// TIA Portal project "ControlPID_FactoryIO" (V16)

(* hardware
DEVICE "S7-1200 station_1"  S7-1200 Station
   slot 0: "Rack_0"  S7-1200 Rack  Rack  V1.0
   slot 1: "PLC_1"  CPU 1214C AC/DC/Rly  6ES7 214-1BG40-0XB0  V4.4
DEVICE "HMI_1"  TP1200 Comfort
   slot 0: "HMI_1"  TP1200 Comfort  6AV2 124-0MC01-0AX0  16.0.0.0
   slot 1: "HMI_RT_1"  TP1200 Comfort  6AV2 124-0MC01-0AX0  16.0.0.0
   slot 5: "HMI_1.IE_CP_1"  PROFINET Interface  16.0.0.0
      slot 1: "PROFINET Interface_1"  PROFINET Interface
         slot 1: "Port_1"  Port
         slot 2: "Port_2"  Port
   slot 7: "HMI_1.MPI/DP_CP_1"  MPI/DP Interface  16.0.0.0
*)

// ===== PLC "PLC_1"  CPU 1214C AC/DC/Rly =====

VAR_GLOBAL   // PLC tag table "Default tag table"
   "Start" AT %I20.0 : Bool;
   "Stop" AT %I20.1 : Bool;
   "Led" AT %Q0.0 : Bool;
   "SP" AT %IW100 : Int;
   "Level Sensor" AT %IW102 : Int;
   "Fill Valve" AT %QW100 : Int;
   "Discharge Valve" AT %QW102 : Int;
   "Display SP" AT %QW104 : Int;
   "Display PV" AT %QW106 : Int;
   "SP(mm)" AT %MD10 : Real;
   "SP(%)" AT %MD14 : Real;
   "PV(mm)" AT %MD18 : Real;
   "PV(%)" AT %MD22 : Real;
   "CV(%)" AT %MD26 : Real;
END_VAR

DATA_BLOCK "Set Point_DB"   // DB1
{ S7_Optimized_Access := 'TRUE' }
VERSION : 0.1
// stored: InstanceOfName Set Point
"Set Point"
BEGIN
END_DATA_BLOCK

DATA_BLOCK "Sensor_DB"   // DB2
{ S7_Optimized_Access := 'TRUE' }
VERSION : 0.1
// stored: InstanceOfName Sensor
"Sensor"
BEGIN
END_DATA_BLOCK

DATA_BLOCK "Output PID_DB"   // DB3
{ S7_Optimized_Access := 'TRUE' }
VERSION : 0.1
// stored: InstanceOfName Output PID
"Output PID"
BEGIN
END_DATA_BLOCK

FUNCTION_BLOCK "Set Point"   // FB1, LAD
{ S7_Optimized_Access := 'TRUE' }
VERSION : 0.1
   VAR_INPUT
      InAnalog : Int;
      LevelMax : Real;
   END_VAR
   VAR_OUTPUT
      "Level(mm)" : Real;
      "Level(%)" : Real;
   END_VAR
   VAR
      Cal : Real;
   END_VAR
BEGIN

REGION Network 1
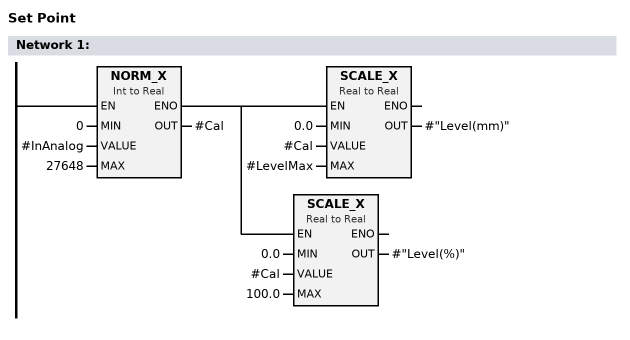
   RUNG wire#powerrail
      { S7_Templates := "[SrcType := Int, DestType := Real]" } Normalize(min := 0, value := #InAnalog, max := 27648, out => #Cal)
      wire#w1
      { S7_Templates := "[SrcType := Real, DestType := Real]" } Scale(min := 0.0, value := #Cal, max := #LevelMax, out => #"Level(mm)")
   END_RUNG
   RUNG wire#w1
      { S7_Templates := "[SrcType := Real, DestType := Real]" } Scale(min := 0.0, value := #Cal, max := 100.0, out => #"Level(%)")
   END_RUNG
   // the same network as SCL:
   #Cal := NORM_X(MIN := 0, VALUE := #InAnalog, MAX := 27648);
   #"Level(mm)" := SCALE_X(MIN := 0.0, VALUE := #Cal, MAX := #LevelMax);
   #"Level(%)" := SCALE_X(MIN := 0.0, VALUE := #Cal, MAX := 100.0);
END_REGION
END_FUNCTION_BLOCK

FUNCTION_BLOCK "Sensor"   // FB2, LAD
{ S7_Optimized_Access := 'TRUE' }
VERSION : 0.1
   VAR_INPUT
      InAnalog : Int;
      LevelMax : Real;
   END_VAR
   VAR_OUTPUT
      "Level(mm)" : Real;
      "Level(%)" : Real;
   END_VAR
   VAR
      Cal : Real;
   END_VAR
BEGIN

REGION Network 1
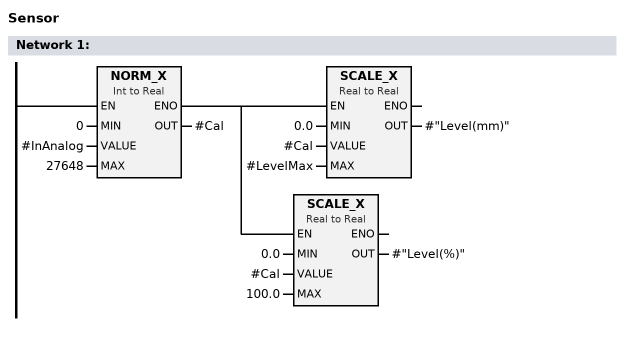
   RUNG wire#powerrail
      { S7_Templates := "[SrcType := Int, DestType := Real]" } Normalize(min := 0, value := #InAnalog, max := 27648, out => #Cal)
      wire#w1
      { S7_Templates := "[SrcType := Real, DestType := Real]" } Scale(min := 0.0, value := #Cal, max := #LevelMax, out => #"Level(mm)")
   END_RUNG
   RUNG wire#w1
      { S7_Templates := "[SrcType := Real, DestType := Real]" } Scale(min := 0.0, value := #Cal, max := 100.0, out => #"Level(%)")
   END_RUNG
   // the same network as SCL:
   #Cal := NORM_X(MIN := 0, VALUE := #InAnalog, MAX := 27648);
   #"Level(mm)" := SCALE_X(MIN := 0.0, VALUE := #Cal, MAX := #LevelMax);
   #"Level(%)" := SCALE_X(MIN := 0.0, VALUE := #Cal, MAX := 100.0);
END_REGION
END_FUNCTION_BLOCK

FUNCTION_BLOCK "Output PID"   // FB3, LAD
{ S7_Optimized_Access := 'TRUE' }
VERSION : 0.1
   VAR_INPUT
      OutputPID : Real;
   END_VAR
   VAR_OUTPUT
      V_Full : Int;
      V_Emty : Int;
   END_VAR
   VAR
      OutputPID_Cal : Real;
      Cal : Real;
      Out_Value : Int;
   END_VAR
BEGIN

REGION Network 1
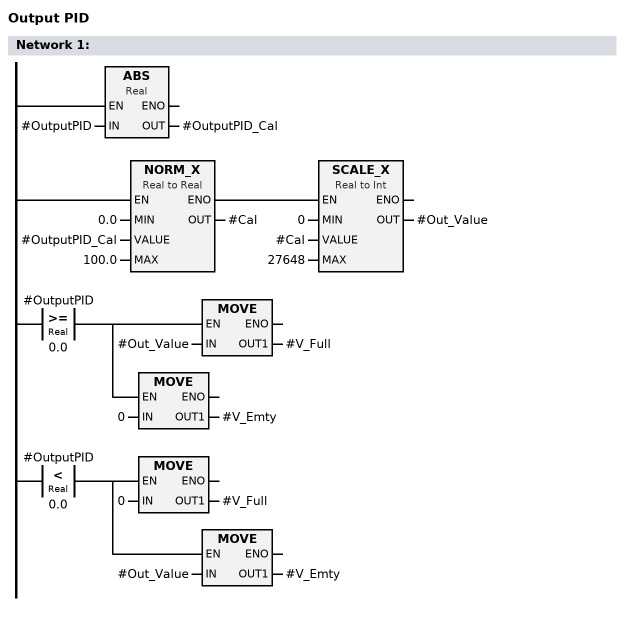
   RUNG wire#powerrail
      { S7_Templates := "SrcType := Real" } Abs(in := #OutputPID, out => #OutputPID_Cal)
   END_RUNG
   RUNG wire#powerrail
      { S7_Templates := "[SrcType := Real, DestType := Real]" } Normalize(min := 0.0, value := #OutputPID_Cal, max := 100.0, out => #Cal)
      { S7_Templates := "[SrcType := Real, DestType := Int]" } Scale(min := 0, value := #Cal, max := 27648, out => #Out_Value)
   END_RUNG
   RUNG wire#powerrail
      { S7_Templates := "SrcType := Real" } GE_Contact(in1 := #OutputPID, in2 := 0.0)
      wire#w1
      Move(in := #Out_Value, out1 => #V_Full)
   END_RUNG
   RUNG wire#w1
      Move(in := 0, out1 => #V_Emty)
   END_RUNG
   RUNG wire#powerrail
      { S7_Templates := "SrcType := Real" } LT_Contact(in1 := #OutputPID, in2 := 0.0)
      wire#w2
      Move(in := 0, out1 => #V_Full)
   END_RUNG
   RUNG wire#w2
      Move(in := #Out_Value, out1 => #V_Emty)
   END_RUNG
   // the same network as SCL:
   #OutputPID_Cal := ABS(#OutputPID);
   #Cal := NORM_X(MIN := 0.0, VALUE := #OutputPID_Cal, MAX := 100.0);
   #Out_Value := SCALE_X(MIN := 0, VALUE := #Cal, MAX := 27648);
   IF #OutputPID >= 0.0 THEN
       #V_Full := #Out_Value;
       #V_Emty := 0;
   END_IF;
   IF #OutputPID < 0.0 THEN
       #V_Full := 0;
       #V_Emty := #Out_Value;
   END_IF;
END_REGION
END_FUNCTION_BLOCK

ORGANIZATION_BLOCK "Main"   // OB1, LAD, ProgramCycle
TITLE = "Main Program Sweep (Cycle)"
{ S7_Optimized_Access := 'TRUE' }
VERSION : 0.1
   VAR_INPUT
      Initial_Call : Bool;   // Initial call of this OB
      Remanence : Bool;   // =True, if remanent data are available
   END_VAR
   VAR_TEMP   // added for the SCL form of the ladder/FBD networks
      _w1 : Bool;
      _w2 : Bool;
   END_VAR
BEGIN

REGION Network 1
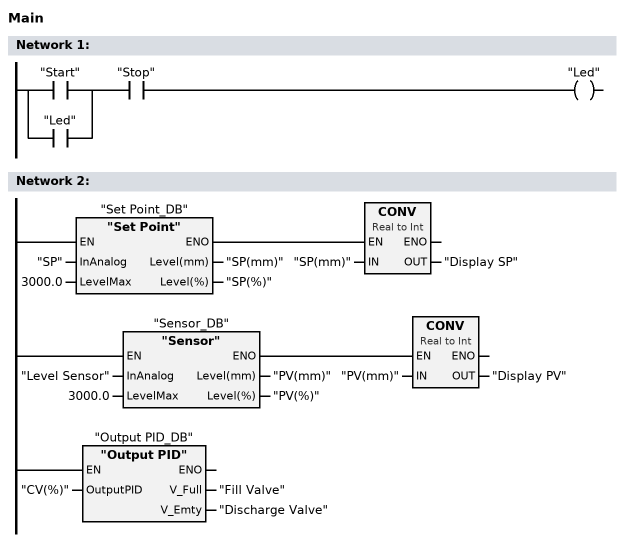
   RUNG wire#powerrail
      Contact( "Start" )
      wire#w1
      Contact( "Stop" )
      Coil( "Led" )
   END_RUNG
   RUNG wire#powerrail
      Contact( "Led" )
   END_RUNG wire#w1
   // the same network as SCL:
   "Led" := ("Start" OR "Led") AND "Stop";
END_REGION

REGION Network 2
   RUNG wire#powerrail
      "Set Point_DB"(InAnalog := "SP", LevelMax := 3000.0, "Level(mm)" => "SP(mm)", "Level(%)" => "SP(%)")
      { S7_Templates := "[SrcType := Real, DestType := Int]" } Convert(in := "SP(mm)", out => "Display SP")
   END_RUNG
   RUNG wire#powerrail
      "Sensor_DB"(InAnalog := "Level Sensor", LevelMax := 3000.0, "Level(mm)" => "PV(mm)", "Level(%)" => "PV(%)")
      { S7_Templates := "[SrcType := Real, DestType := Int]" } Convert(in := "PV(mm)", out => "Display PV")
   END_RUNG
   RUNG wire#powerrail
      "Output PID_DB"(OutputPID := "CV(%)", V_Full => "Fill Valve", V_Emty => "Discharge Valve")
   END_RUNG
   // the same network as SCL:
   "Set Point_DB"(InAnalog := "SP",   // "Set Point"
                  LevelMax := 3000.0,
                  "Level(mm)" => "SP(mm)",
                  "Level(%)" => "SP(%)",
                  ENO => #_w1);
   IF #_w1 THEN "Display SP" := REAL_TO_INT("SP(mm)"); END_IF;
   "Sensor_DB"(InAnalog := "Level Sensor",   // "Sensor"
               LevelMax := 3000.0,
               "Level(mm)" => "PV(mm)",
               "Level(%)" => "PV(%)",
               ENO => #_w2);
   IF #_w2 THEN "Display PV" := REAL_TO_INT("PV(mm)"); END_IF;
   "Output PID_DB"(OutputPID := "CV(%)", V_Full => "Fill Valve", V_Emty => "Discharge Valve");   // "Output PID"
END_REGION
END_ORGANIZATION_BLOCK

ORGANIZATION_BLOCK "Cyclic interrupt"   // OB30, LAD, CyclicInterrupt
{ S7_Optimized_Access := 'TRUE' }
VERSION : 0.1
   VAR_INPUT
      Initial_Call : Bool;   // Initial call of this OB
      Event_Count : Int;   // Events discarded
   END_VAR
BEGIN

REGION Network 1
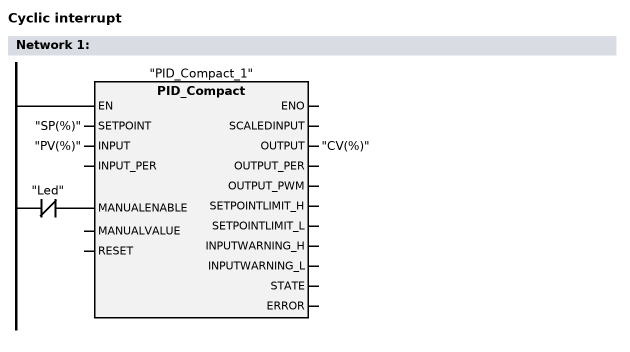
   "PID_Compact_1"(Setpoint := "SP(%)", Input := "PV(%)", ManualEnable := NOT "Led", Output => "CV(%)");   // PID_Compact
END_REGION
END_ORGANIZATION_BLOCK

(* ===== HMI "HMI_RT_1" =====
system functions are stored by id; their names below are inferred from use
connection "HMI_Connection_1": ETHERNET, S7_1200_OMS

HMI tags "Default tag table"
   "Tag_ScreenNumber" : UInt, internal
   "SP(mm)" : Real = PLC "SP(mm)" AT %MD10, 1 s
   "PV(mm)" : Real = PLC "PV(mm)" AT %MD18, 1 s
   "SP(%)" : Real = PLC "SP(%)" AT %MD14, 1 s
   "PV(%)" : Real = PLC "PV(%)" AT %MD22, 1 s
   "CV(%)" : Real = PLC "CV(%)" AT %MD26, 1 s
   "Fill Valve" : Int = PLC "Fill Valve" AT %QW100, 1 s
   "Discharge Valve" : Int = PLC "Discharge Valve" AT %QW102, 1 s

screen "Root screen" 1280x740, template "Template_1"
   on GenerateScreen: SetTag("Tag_ScreenNumber", 1)
   IOField "I/O field_1" at 17,27 size 124x43; FormatPattern 9999.99; Unit mm
      ProcessValue <- "SP(mm)"
   Group "Group" at 288,109 size 136x163
   IOField "I/O field_2" at 52,75 size 81x36; FormatPattern 99.99; Unit %
      ProcessValue <- "SP(%)"
   TextField "Text field_2" at 21,2 size 36x25; Text 'SP:'
   IOField "I/O field_3" at 25,218 size 116x43; FormatPattern 9999.99; Unit mm
      ProcessValue <- "PV(mm)"
   IOField "I/O field_4" at 52,266 size 81x36; FormatPattern 99.99; Unit %
      ProcessValue <- "PV(%)"
   TextField "Text field_3" at 21,193 size 36x25; Text 'PV:'
   IOField "I/O field_5" at 597,183 size 112x43; FormatPattern s99.99; Unit %
      ProcessValue <- "CV(%)"
   IOField "I/O field_6" at 620,231 size 81x36; FormatPattern 99999
      ProcessValue <- "Fill Valve"
   TextField "Text field_4" at 589,158 size 36x25; Text 'CV:'
   IOField "I/O field_7" at 620,285 size 81x36; FormatPattern 99999
      ProcessValue <- "Discharge Valve"
   TextField "Text field_5" at 508,292 size 117x25; Text 'V Discharge'
   TextField "Text field_6" at 537,241 size 52x25; Text 'V Fill'
   TrendView "Trend view_1" at 711,43 size 568x515
   TextField "Text field_1" at 295,118 size 129x46; Text 'PID CONTROLLER'

Template "Template_1" 1280x740
   Button "Exit" at 1200,679 size 78x59; TextOff 'Exit'; PictureOff "ExitRuntime_TP1200_Comfort_TR"; PictureOn "ExitRuntime_TP1200_Comfort_TR"
      on Release: StopRuntime(0)
   Button "Template_Button" at 1120,679 size 78x59; TextOff 'Text'
   Button "Template_Button_1" at 1040,679 size 78x59; TextOff 'Text'
   Button "Template_Button_2" at 960,679 size 78x59; TextOff 'Text'
   Button "Template_Button_3" at 880,679 size 78x59; TextOff 'Text'
   Button "Template_Button_4" at 800,679 size 78x59; TextOff 'Text'
   Button "Template_Button_5" at 720,679 size 78x59; TextOff 'Text'
   Button "Template_Button_6" at 640,679 size 78x59; TextOff 'Text'
   Button "Template_Button_7" at 561,679 size 78x59; TextOff 'Text'
   Button "Template_Button_8" at 481,679 size 78x59; TextOff 'Text'
   Button "Template_Button_9" at 401,679 size 78x59; TextOff 'Text'
   Button "Template_Button_10" at 321,679 size 78x59; TextOff 'Text'
   Button "Template_Button_11" at 241,679 size 78x59; TextOff 'Text'
   Button "Template_Button_12" at 161,679 size 78x59; TextOff 'Text'
   Button "Alarms" at 81,679 size 78x59; TextOff 'Alarms'; PictureOff "AlarmDisplay_TP1200_Comfort_TR"; PictureOn "AlarmDisplay_TP1200_Comfort_TR"
      on Release: function_ef3f5d25("Alarm window_Unacknowledged", -1)
   Button "Start screen" at 1,679 size 78x59; TextOff 'Start screen'; PictureOff "NavigateHome_TP1200_Comfort_TR"; PictureOn "NavigateHome_TP1200_Comfort_TR"
      on Release: ActivateScreen("Root screen", 0)
*)